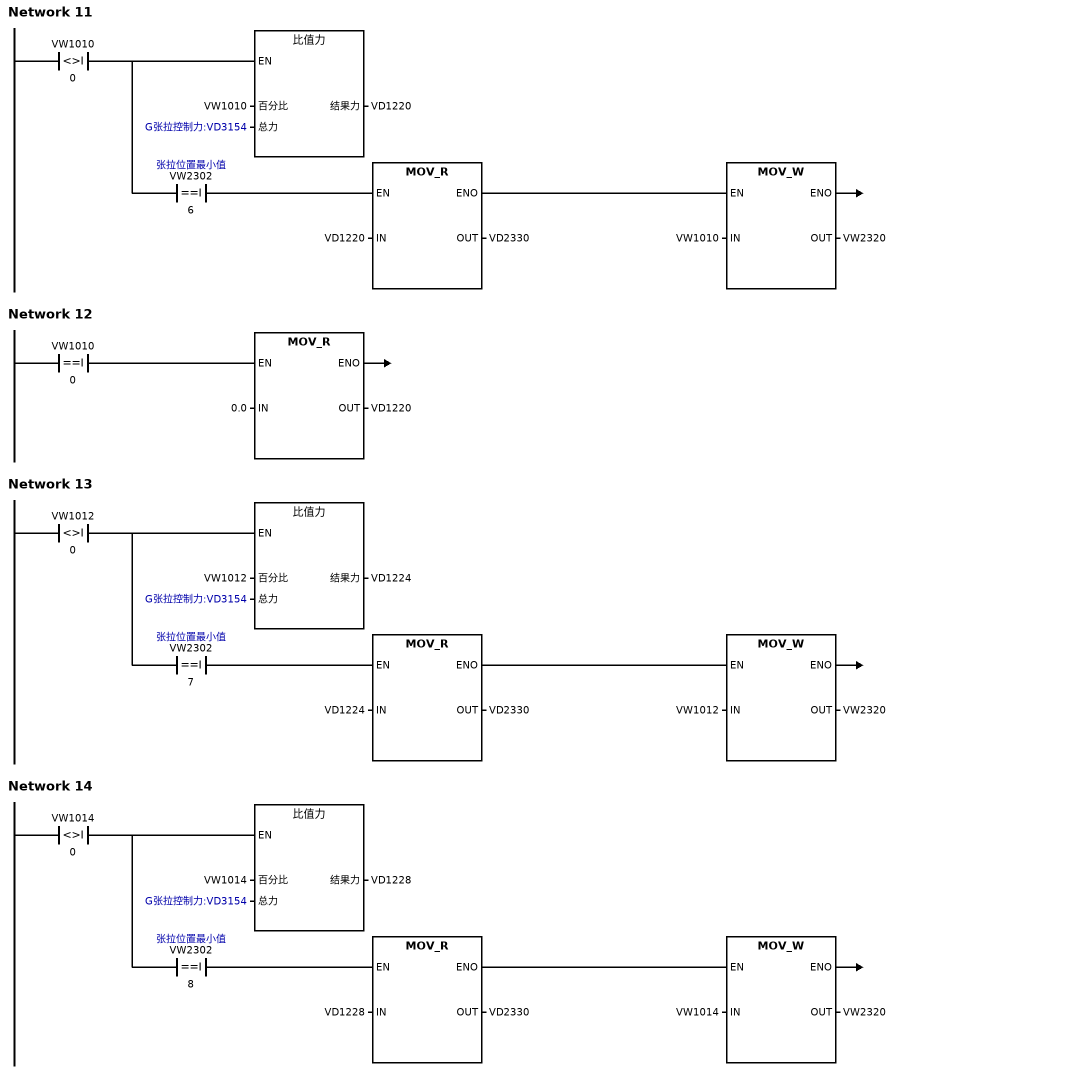
[picture p72: SBR24 networks 11-14]
Network 11
LDW<>  VW1010, 0
CALL   比值力:SBR25, VW1010, G张拉控制力:VD3154, VD1220
AW=    张拉位置最小值:VW2302, 6
MOVR   VD1220, VD2330
AENO
MOVW   VW1010, VW2320
Network 12
LDW=   VW1010, 0
MOVR   0.0, VD1220
Network 13
LDW<>  VW1012, 0
CALL   比值力:SBR25, VW1012, G张拉控制力:VD3154, VD1224
AW=    张拉位置最小值:VW2302, 7
MOVR   VD1224, VD2330
AENO
MOVW   VW1012, VW2320
Network 14
LDW<>  VW1014, 0
CALL   比值力:SBR25, VW1014, G张拉控制力:VD3154, VD1228
AW=    张拉位置最小值:VW2302, 8
MOVR   VD1228, VD2330
AENO
MOVW   VW1014, VW2320
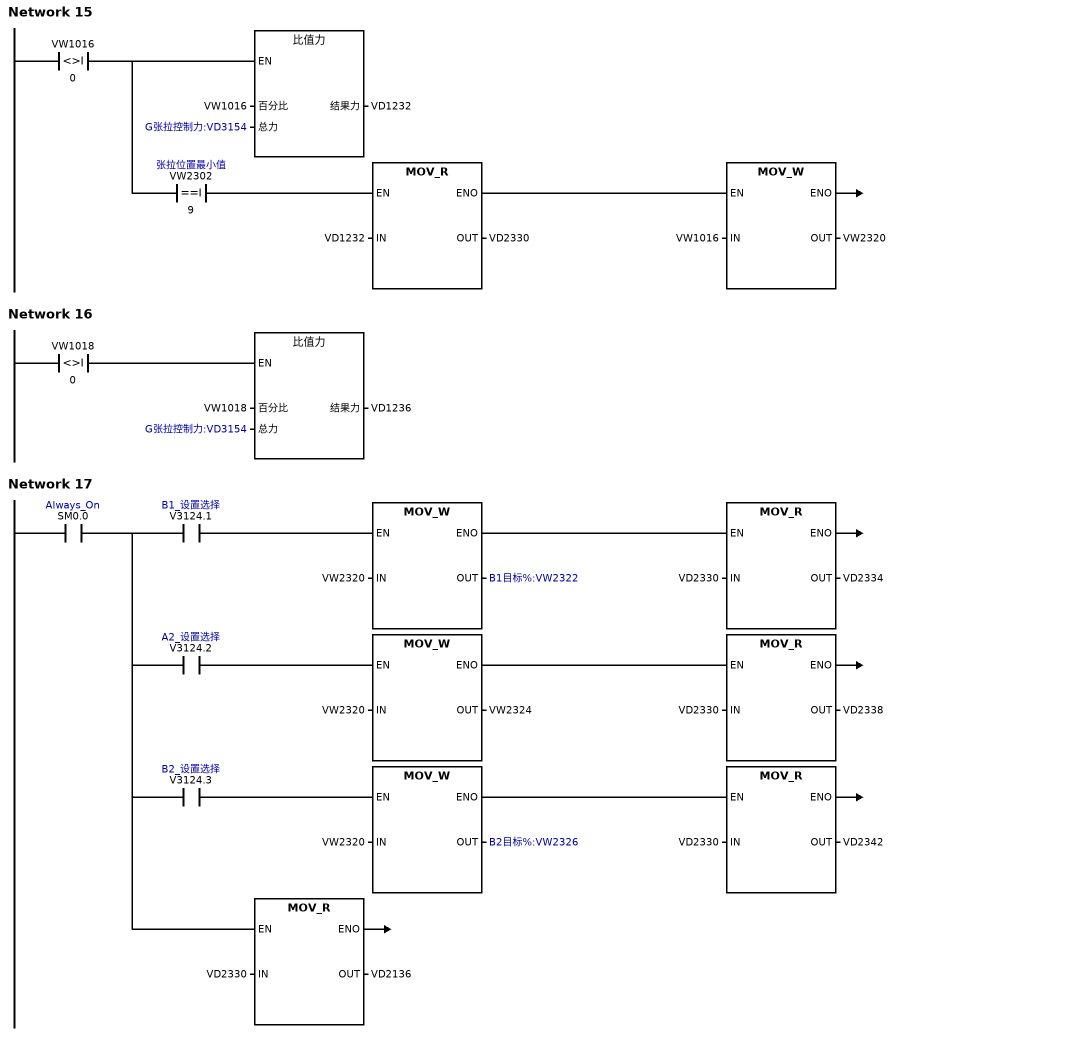
Network 15
LDW<>  VW1016, 0
CALL   比值力:SBR25, VW1016, G张拉控制力:VD3154, VD1232
AW=    张拉位置最小值:VW2302, 9
MOVR   VD1232, VD2330
AENO
MOVW   VW1016, VW2320
Network 16
LDW<>  VW1018, 0
CALL   比值力:SBR25, VW1018, G张拉控制力:VD3154, VD1236
Network 17
LD     Always_On:SM0.0
LPS
A      B1_设置选择:V3124.1
MOVW   VW2320, B1目标%:VW2322
AENO
MOVR   VD2330, VD2334
LRD
A      A2_设置选择:V3124.2
MOVW   VW2320, VW2324
AENO
MOVR   VD2330, VD2338
LRD
A      B2_设置选择:V3124.3
MOVW   VW2320, B2目标%:VW2326
AENO
MOVR   VD2330, VD2342
LPP
MOVR   VD2330, VD2136
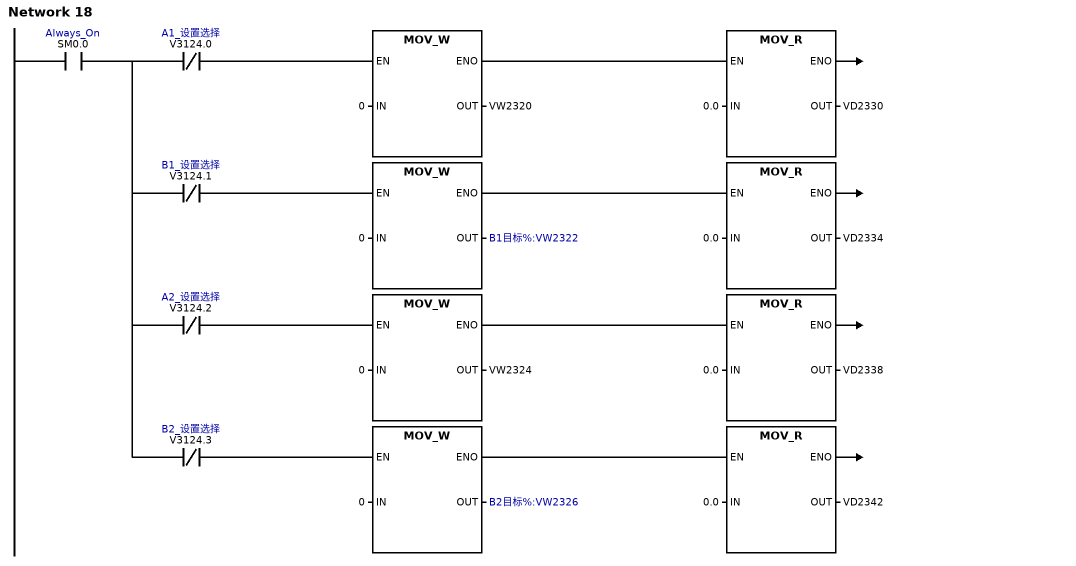
Network 18
LD     Always_On:SM0.0
LPS
AN     A1_设置选择:V3124.0
MOVW   0, VW2320
AENO
MOVR   0.0, VD2330
LRD
AN     B1_设置选择:V3124.1
MOVW   0, B1目标%:VW2322
AENO
MOVR   0.0, VD2334
LRD
AN     A2_设置选择:V3124.2
MOVW   0, VW2324
AENO
MOVR   0.0, VD2338
LPP
AN     B2_设置选择:V3124.3
MOVW   0, B2目标%:VW2326
AENO
MOVR   0.0, VD2342
END_SUBROUTINE_BLOCK

SUBROUTINE_BLOCK 比值力:SBR25
TITLE=子程序注释
VAR_INPUT
百分比:INT;	// LW0 
总力:REAL;	// LD2 
END_VAR
VAR_OUTPUT
结果力:REAL;	// LD6 
END_VAR
VAR
中间力:REAL;	// LD10 
END_VAR
BEGIN
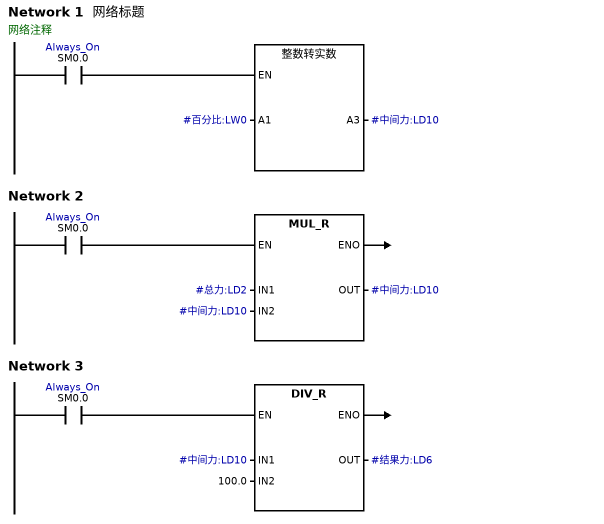
Network 1 // 网络标题
// 网络注释
LD     Always_On:SM0.0
CALL   整数转实数:SBR5, #百分比:LW0, #中间力:LD10
Network 2
LD     Always_On:SM0.0
*R     #总力:LD2, #中间力:LD10
Network 3
LD     Always_On:SM0.0
MOVR   #中间力:LD10, #结果力:LD6
/R     100.0, #结果力:LD6
END_SUBROUTINE_BLOCK

SUBROUTINE_BLOCK F_AK_B:SBR26
TITLE=子程序注释
VAR_INPUT
k1:INT;	// LW0 
XSA1:REAL;	// LD2 
XSB1:REAL;	// LD6 
END_VAR
VAR_OUTPUT
F1:REAL;	// LD10 
END_VAR
VAR
ZJ:REAL;	// LD14 
END_VAR
BEGIN
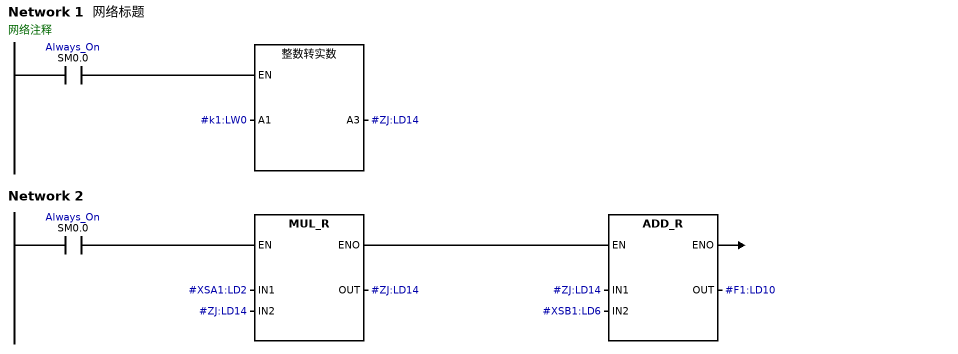
Network 1 // 网络标题
// 网络注释
LD     Always_On:SM0.0
CALL   整数转实数:SBR5, #k1:LW0, #ZJ:LD14
Network 2
LD     Always_On:SM0.0
*R     #XSA1:LD2, #ZJ:LD14
AENO
MOVR   #ZJ:LD14, #F1:LD10
+R     #XSB1:LD6, #F1:LD10
END_SUBROUTINE_BLOCK

SUBROUTINE_BLOCK 波动滤波:SBR27
TITLE=子程序注释
VAR_INPUT
dq:INT;	// LW0 
jiyi:INT;	// LW2 
py:INT;	// LW4 
END_VAR
VAR_OUTPUT
sj:INT;	// LW6 
END_VAR
VAR
add1:INT;	// LW8 
sub1:INT;	// LW10 
END_VAR
BEGIN
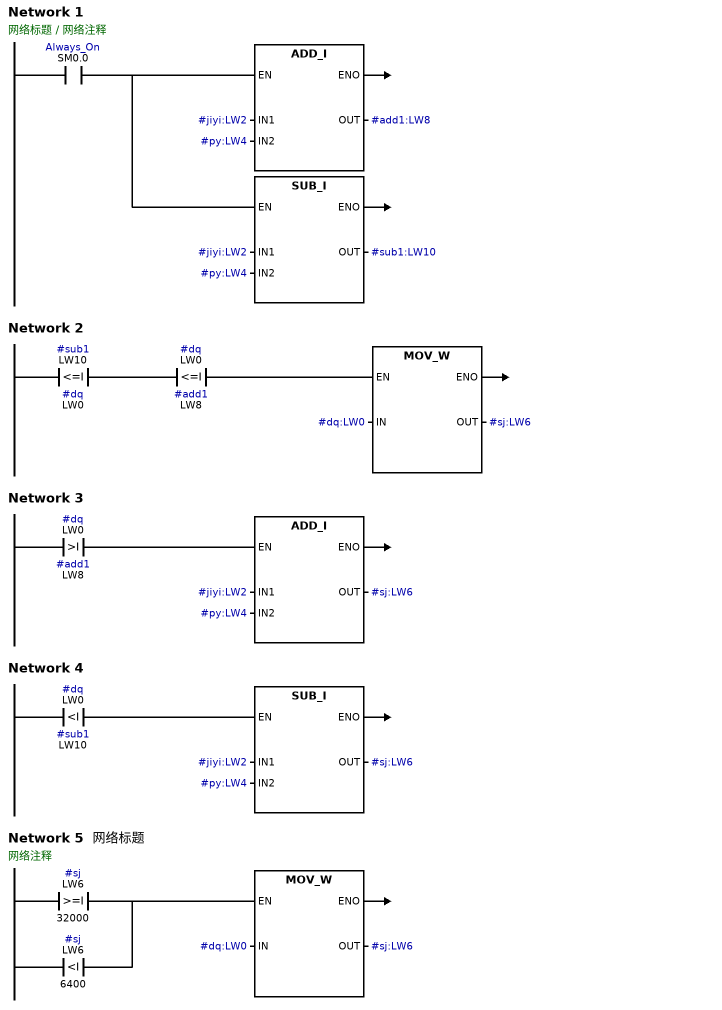
Network 1
// 网络标题
// 网络注释
LD     Always_On:SM0.0
MOVW   #jiyi:LW2, #add1:LW8
+I     #py:LW4, #add1:LW8
MOVW   #jiyi:LW2, #sub1:LW10
-I     #py:LW4, #sub1:LW10
Network 2
LDW<=  #sub1:LW10, #dq:LW0
AW<=   #dq:LW0, #add1:LW8
MOVW   #dq:LW0, #sj:LW6
Network 3
LDW>   #dq:LW0, #add1:LW8
MOVW   #jiyi:LW2, #sj:LW6
+I     #py:LW4, #sj:LW6
Network 4
LDW<   #dq:LW0, #sub1:LW10
MOVW   #jiyi:LW2, #sj:LW6
-I     #py:LW4, #sj:LW6
Network 5 // 网络标题
// 网络注释
LDW>=  #sj:LW6, 32000
OW<    #sj:LW6, 6400
MOVW   #dq:LW0, #sj:LW6
END_SUBROUTINE_BLOCK

SUBROUTINE_BLOCK 取张拉时间:SBR28
TITLE=子程序注释
BEGIN
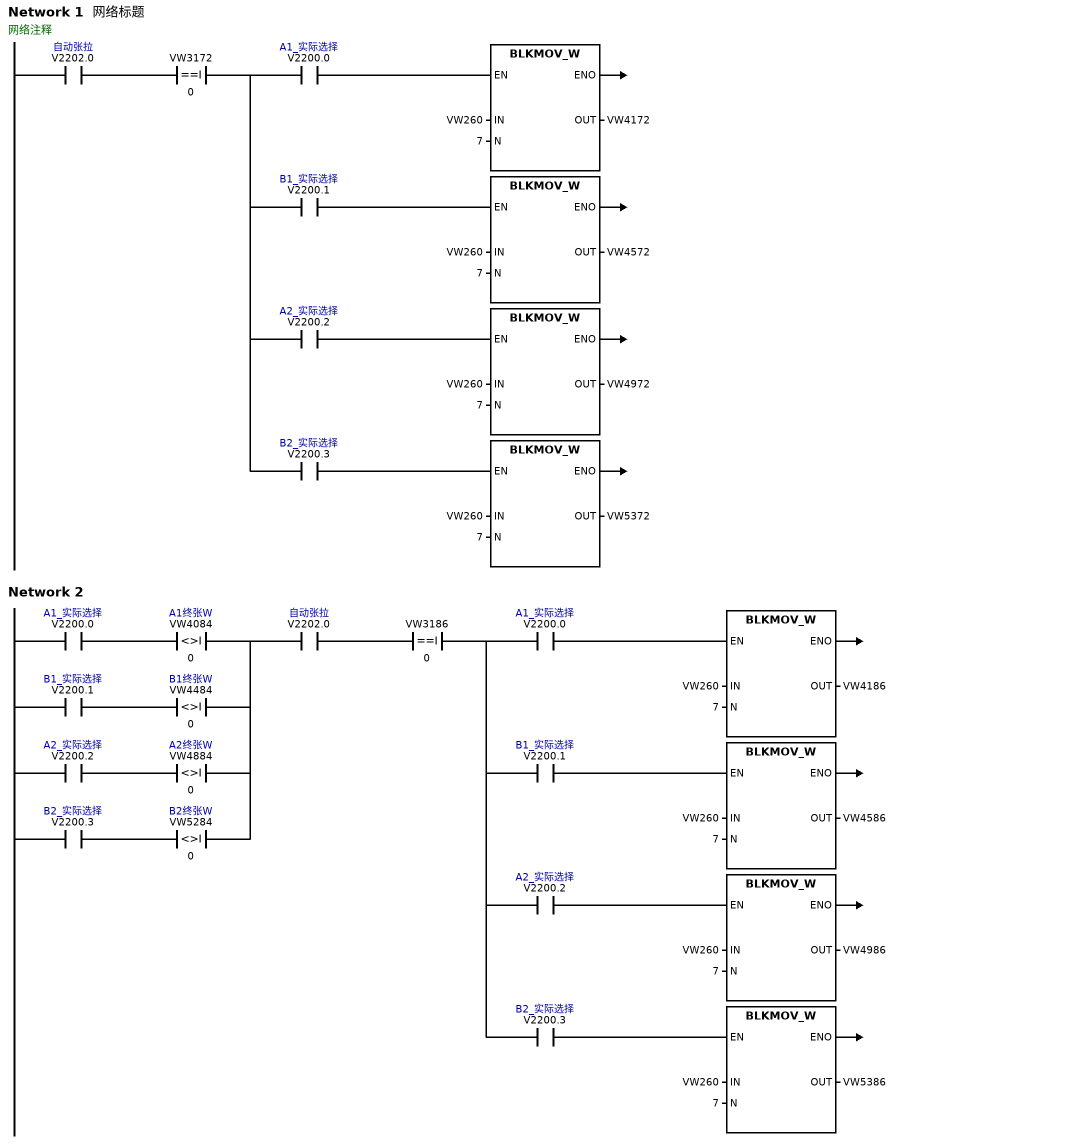
Network 1 // 网络标题
// 网络注释
LD     自动张拉:V2202.0
AW=    VW3172, 0
LPS
A      A1_实际选择:V2200.0
BMW    VW260, VW4172, 7
LRD
A      B1_实际选择:V2200.1
BMW    VW260, VW4572, 7
LRD
A      A2_实际选择:V2200.2
BMW    VW260, VW4972, 7
LPP
A      B2_实际选择:V2200.3
BMW    VW260, VW5372, 7
Network 2
LD     A1_实际选择:V2200.0
AW<>   A1终张W:VW4084, 0
LD     B1_实际选择:V2200.1
AW<>   B1终张W:VW4484, 0
OLD
LD     A2_实际选择:V2200.2
AW<>   A2终张W:VW4884, 0
OLD
LD     B2_实际选择:V2200.3
AW<>   B2终张W:VW5284, 0
OLD
A      自动张拉:V2202.0
AW=    VW3186, 0
LPS
A      A1_实际选择:V2200.0
BMW    VW260, VW4186, 7
LRD
A      B1_实际选择:V2200.1
BMW    VW260, VW4586, 7
LRD
A      A2_实际选择:V2200.2
BMW    VW260, VW4986, 7
LPP
A      B2_实际选择:V2200.3
BMW    VW260, VW5386, 7
END_SUBROUTINE_BLOCK

SUBROUTINE_BLOCK 主机与电脑:SBR29
TITLE=子程序注释
BEGIN
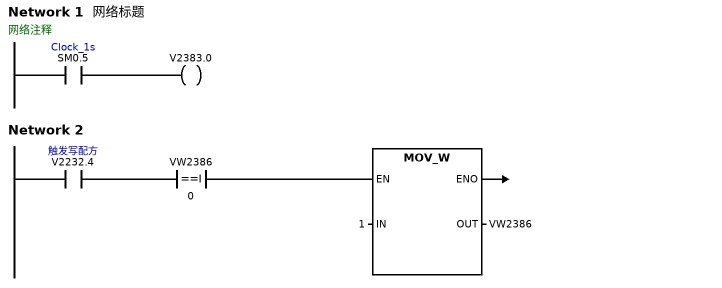
Network 1 // 网络标题
// 网络注释
LD     Clock_1s:SM0.5
=      V2383.0
Network 2
LD     触发写配方:V2232.4
AW=    VW2386, 0
MOVW   1, VW2386
END_SUBROUTINE_BLOCK

SUBROUTINE_BLOCK 频率给定:SBR30
TITLE=子程序注释
BEGIN
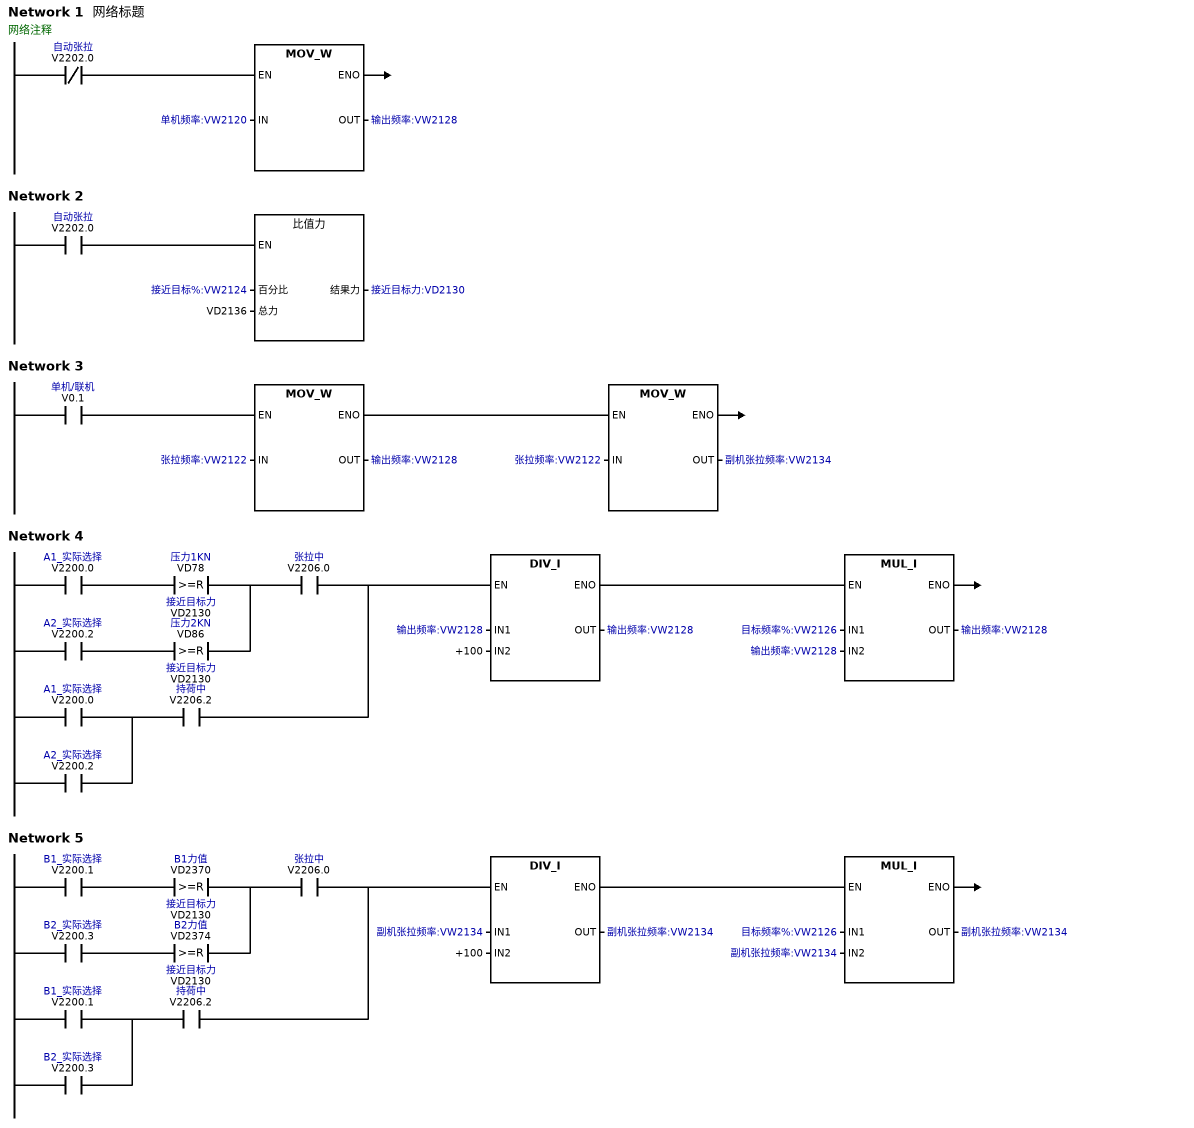
Network 1 // 网络标题
// 网络注释
LDN    自动张拉:V2202.0
MOVW   单机频率:VW2120, 输出频率:VW2128
Network 2
LD     自动张拉:V2202.0
CALL   比值力:SBR25, 接近目标%:VW2124, VD2136, 接近目标力:VD2130
Network 3
LD     单机/联机:V0.1
MOVW   张拉频率:VW2122, 输出频率:VW2128
AENO
MOVW   张拉频率:VW2122, 副机张拉频率:VW2134
Network 4
LD     A1_实际选择:V2200.0
AR>=   压力1KN:VD78, 接近目标力:VD2130
LD     A2_实际选择:V2200.2
AR>=   压力2KN:VD86, 接近目标力:VD2130
OLD
A      张拉中:V2206.0
LD     A1_实际选择:V2200.0
O      A2_实际选择:V2200.2
A      持荷中:V2206.2
OLD
/I     +100, 输出频率:VW2128
AENO
*I     目标频率%:VW2126, 输出频率:VW2128
Network 5
LD     B1_实际选择:V2200.1
AR>=   B1力值:VD2370, 接近目标力:VD2130
LD     B2_实际选择:V2200.3
AR>=   B2力值:VD2374, 接近目标力:VD2130
OLD
A      张拉中:V2206.0
LD     B1_实际选择:V2200.1
O      B2_实际选择:V2200.3
A      持荷中:V2206.2
OLD
/I     +100, 副机张拉频率:VW2134
AENO
*I     目标频率%:VW2126, 副机张拉频率:VW2134
END_SUBROUTINE_BLOCK

INTERRUPT_BLOCK 定时:INT10
TITLE=中断程序注释
BEGIN
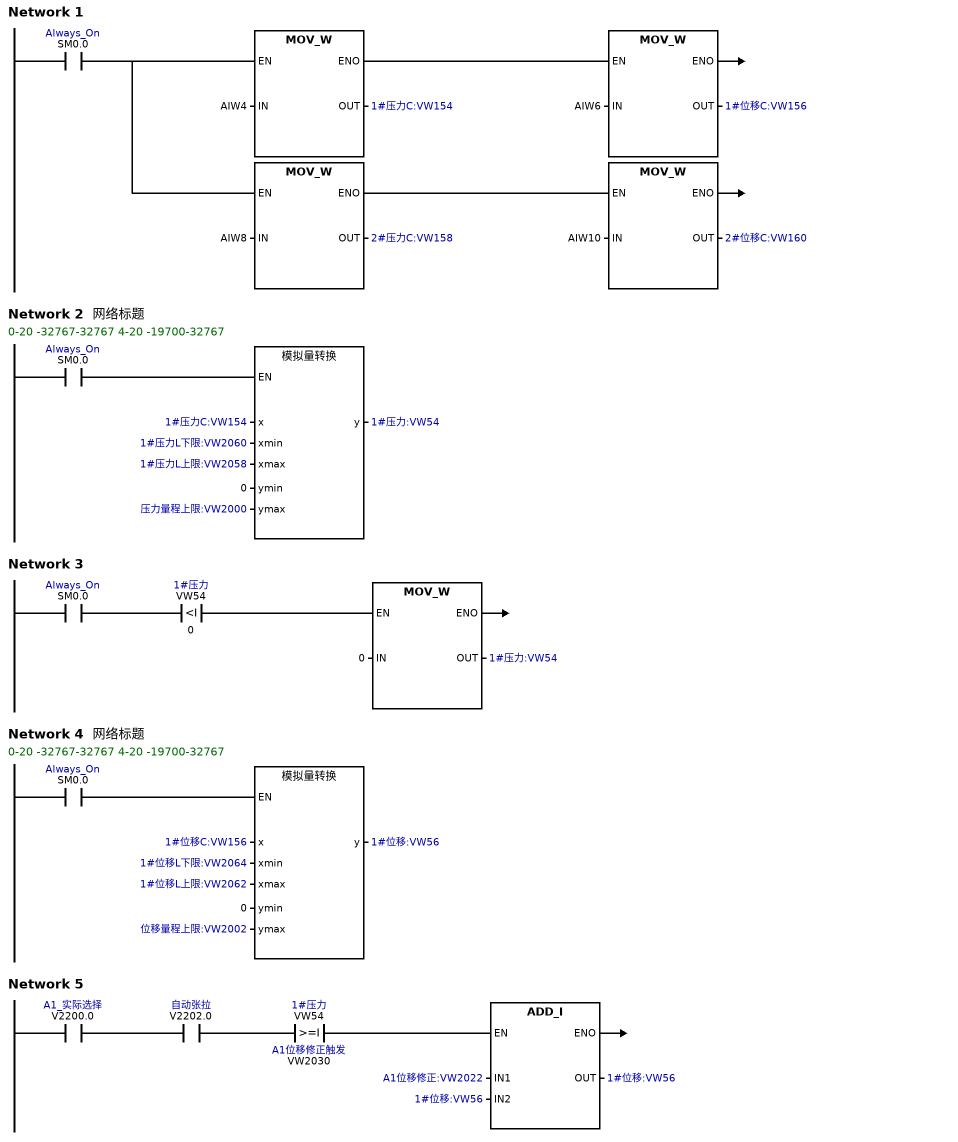
Network 1
LD     Always_On:SM0.0
LPS
MOVW   AIW4, 1#压力C:VW154
AENO
MOVW   AIW6, 1#位移C:VW156
LPP
MOVW   AIW8, 2#压力C:VW158
AENO
MOVW   AIW10, 2#位移C:VW160
Network 2 // 网络标题
// 0-20 -32767-32767 4-20 -19700-32767
LD     Always_On:SM0.0
CALL   模拟量转换:SBR4, 1#压力C:VW154, 1#压力L下限:VW2060, 1#压力L上限:VW2058, 0, 压力量程上限:VW2000, 1#压力:VW54
Network 3
LD     Always_On:SM0.0
AW<    1#压力:VW54, 0
MOVW   0, 1#压力:VW54
Network 4 // 网络标题
// 0-20 -32767-32767 4-20 -19700-32767
LD     Always_On:SM0.0
CALL   模拟量转换:SBR4, 1#位移C:VW156, 1#位移L下限:VW2064, 1#位移L上限:VW2062, 0, 位移量程上限:VW2002, 1#位移:VW56
Network 5
LD     A1_实际选择:V2200.0
A      自动张拉:V2202.0
AW>=   1#压力:VW54, A1位移修正触发:VW2030
+I     A1位移修正:VW2022, 1#位移:VW56
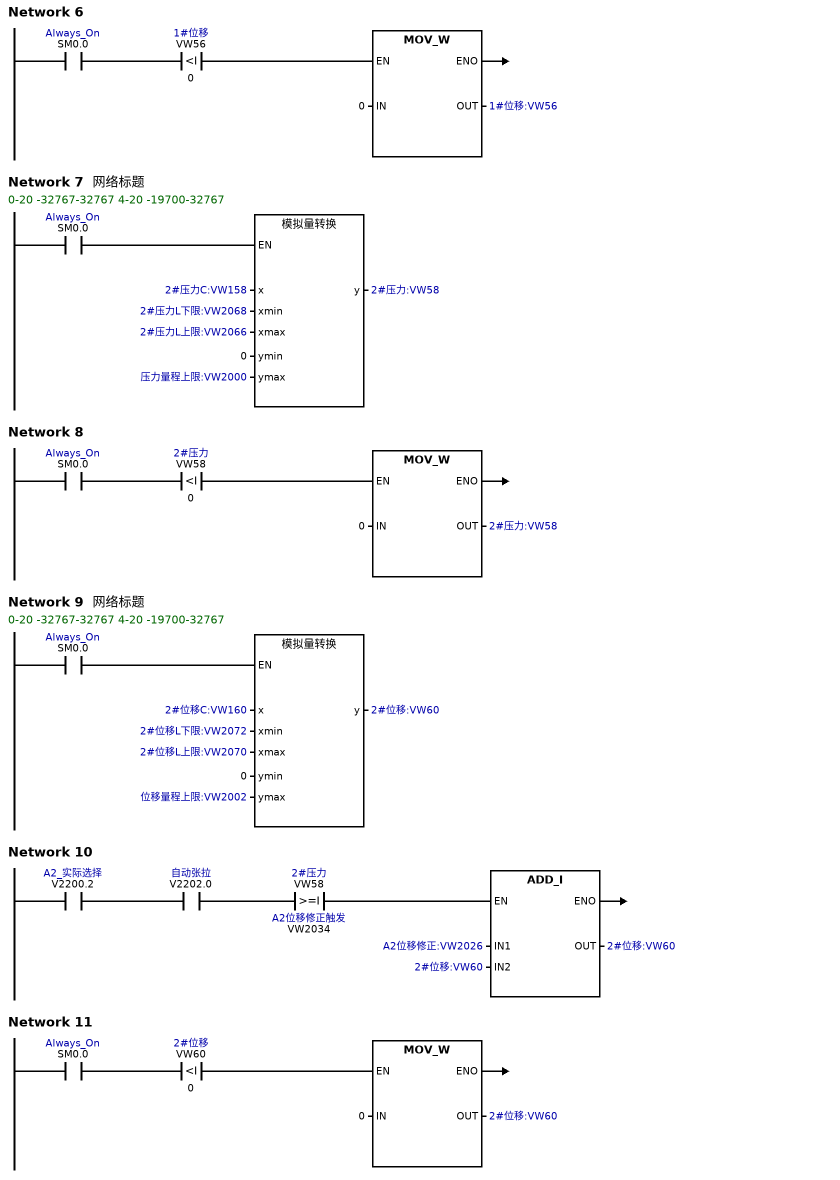
Network 6
LD     Always_On:SM0.0
AW<    1#位移:VW56, 0
MOVW   0, 1#位移:VW56
Network 7 // 网络标题
// 0-20 -32767-32767 4-20 -19700-32767
LD     Always_On:SM0.0
CALL   模拟量转换:SBR4, 2#压力C:VW158, 2#压力L下限:VW2068, 2#压力L上限:VW2066, 0, 压力量程上限:VW2000, 2#压力:VW58
Network 8
LD     Always_On:SM0.0
AW<    2#压力:VW58, 0
MOVW   0, 2#压力:VW58
Network 9 // 网络标题
// 0-20 -32767-32767 4-20 -19700-32767
LD     Always_On:SM0.0
CALL   模拟量转换:SBR4, 2#位移C:VW160, 2#位移L下限:VW2072, 2#位移L上限:VW2070, 0, 位移量程上限:VW2002, 2#位移:VW60
Network 10
LD     A2_实际选择:V2200.2
A      自动张拉:V2202.0
AW>=   2#压力:VW58, A2位移修正触发:VW2034
+I     A2位移修正:VW2026, 2#位移:VW60
Network 11
LD     Always_On:SM0.0
AW<    2#位移:VW60, 0
MOVW   0, 2#位移:VW60
END_INTERRUPT_BLOCK
